{attribute 'linkalways'} 
{attribute 'no_explicit_call' := 'This FB is a CLASS and must be accessed using methods or properties'}
{attribute 'enable_dynamic_creation'}
FUNCTION_BLOCK Node_F_VN_AppendToContainer_TcVnPoint2_LREAL EXTENDS VisionNode
VAR
    aElement : _TcVnPoint2_LREAL;
    ipContainer : _ITcVnContainer;
    hrPrev : _HRESULT(S_OK);
	hresult : _HRESULT(S_OK);
END_VAR

METHOD PUBLIC  Clone : I_Node
VAR
	pNode : POINTER TO Node_F_VN_AppendToContainer_TcVnPoint2_LREAL;
END_VAR
pNode := __NEW(Node_F_VN_AppendToContainer_TcVnPoint2_LREAL);
Clone := pNode^;
END_METHOD

METHOD FB_init : BOOL
VAR_INPUT
	bInitRetains : BOOL; // if TRUE, the retain variables are initialized (warm start / cold start)
	bInCopyCode : BOOL;  // if TRUE, the instance afterwards gets moved into the copy code (online change)
END_VAR
AddInput('aElement', aElement);
AddInput('ipContainer', ipContainer);
AddInput('hrPrev', hrPrev);
AddOutput('ipContainer', ipContainer);
AddOutput('hresult',hresult);
END_METHOD

METHOD PROTECTED OnExecute
hresult.Value := F_VN_AppendToContainer_TcVnPoint2_LREAL(
    aElement := aElement.Value,
	ipContainer := ipContainer.Value,
	hrPrev:= hrPrev.Value);
END_METHOD

METHOD PUBLIC PreExecutionCheck
VAR_INPUT
	Check : I_PreExecutionChecks;
END_VAR
Check.IsTrue(ipContainer.IsValid, 'ipContainer must be a valid container');
Check.IsTrue(ipContainer.IsType(TC_GLOBAL_CONST_LIST.ContainerType_Vector_TcVnPoint2_LREAL), 'ipContainer contains incorrect type');
END_METHOD

END_FUNCTION_BLOCK

(* stored: Version 1.1.0.1, ProductVersion 3.1.4026.13
   POU Node_F_VN_AppendToContainer_TcVnPoint2_LREAL: Id {7d5fd228-15d6-41ae-846c-b3e1887b136b}, SpecialFunc None
   Folder Constructor: Id {7cd5c79f-2126-4ba7-ab07-bd950dc2979f}
   Method Clone: Id {34d6cc21-18df-4148-9511-22d80af8d9fa}
   Method FB_init: Id {9e1bcb3e-f8a4-42cc-a61c-14ba1a1b07d2}
   Method OnExecute: Id {2ef157e5-fcf7-4aa5-8d6c-b3d1bd6bc116}
   Method PreExecutionCheck: Id {bc5b20cc-d896-4f04-a413-394ce4784b12} *)
